// TIA Portal V19 export
TYPE "PosFbk_Encoder_TEL81"
// stored: Access Published
   STRUCT
      IN : Struct
         ZSW2_ENC : Struct
            b_08 : Bool;
            CTRL_REQ : Bool;   // Control requested: 0=No control by the PLC requested, 1=Control by the PLC requested
            b_10 : Bool;
            b_11 : Bool;
            SoL_0 : Bool;   // Encoder’s Sign-of-Life (not relevant)
            SoL_1 : Bool;   // Encoder’s Sign-of-Life (not relevant)
            SoL_2 : Bool;   // Encoder’s Sign-of-Life (not relevant)
            SoL_3 : Bool;   // Encoder’s Sign-of-Life (not relevant)
            b_00 : Bool;
            b_01 : Bool;
            b_02 : Bool;
            b_03 : Bool;
            b_04 : Bool;
            b_05 : Bool;
            b_06 : Bool;
            b_07 : Bool;
         END_STRUCT;
         G1_ZSW : Struct
            b_08 : Bool;
            b_09 : Bool;
            b_10 : Bool;
            REQ_ERR_ACK : Bool;   // Requirement of error acknowledgement detected: 0=No return acknowledgement of encoder error1, =Requirement of error acknowledgement detected
            PSET_STS : Bool;   // Status of the Preset function (set/shift of home position executed): 0=No Preset function active, 1=Preset function is runFeedback based on G1_STW bit12:
            TRM_ABS_POS : Bool;   // Transmission of absolute position value: 0=No transmission, 1=Position value is output in G1_XIST2
            PARK_MODE : Bool;   // Park mode activated: 0=Normal operation, 1=Park mode activatedFeedback based on G1_STW bit14:No output of position data G1_XIST1and G1_XIST2
            ENC_ERR : Bool;   // Encoder error: 0=No error, 1=ErrorThe error code is output in G1_XIST2
            b_00 : Bool;
            b_01 : Bool;
            b_02 : Bool;
            b_03 : Bool;
            b_04 : Bool;
            b_05 : Bool;
            b_06 : Bool;
            b_07 : Bool;
         END_STRUCT;
         G1_XIST1 : DInt;
         G1_XIST2 : DInt;
      END_STRUCT;
      OUT : Struct
         STW2_ENC : Struct
            b_08 : Bool;
            b_09 : Bool;
            PLC_CTRL : Bool;   // Control by PLC: 0=No control by the PLC, 1 =Control by the PLCEnables the PLC by using controlwords to activate / deactivate encoder functions
            b_11 : Bool;
            SoL_0 : Bool;   // Master’s Sign-of-Life (not relevant)
            SoL_1 : Bool;   // Master’s Sign-of-Life (not relevant)
            SoL_2 : Bool;   // Master’s Sign-of-Life (not relevant)
            SoL_3 : Bool;   // Master’s Sign-of-Life (not relevant)
            b_00 : Bool;
            b_01 : Bool;
            b_02 : Bool;
            b_03 : Bool;
            b_04 : Bool;
            b_05 : Bool;
            b_06 : Bool;
            FLT_ACK : Bool;   // Fault acknowledge: Error-buffer handling not supported
         END_STRUCT;
         G1_STW : Struct
            b_08 : Bool;
            b_09 : Bool;
            b_10 : Bool;
            PSET_MODE : Bool;   // 0=ABS 1=REL
            PSET_ACT : Bool;   // Activate preset value
            POS_REQ : Bool;   // Request for the absolute positionvalue
            PARK_MODE : Bool;   // Activate park mode 0=Normal operation, 1=Activate park mode
            ERR_ACK : Bool;   // Acknowledging a sensor error 0=Encoder error message notacknowledged by PLC, 1=Encoder error message acknowledged by the PLC
            b_00 : Bool;
            b_01 : Bool;
            b_02 : Bool;
            b_03 : Bool;
            b_04 : Bool;
            b_05 : Bool;
            b_06 : Bool;
            b_07 : Bool;
         END_STRUCT;
      END_STRUCT;
   END_STRUCT;
END_TYPE
